VAR_GLOBAL
	DAU : ARRAY [1..100] OF DAU; //Instantiate 100 DAU's  This can be made higher if we think that 1 system will ever have more than 100 DAU's
END_VAR

(* stored: Version 1.1.0.1, ProductVersion 3.1.4022.12
   GVL GVL_DUA: Id {964d5aa3-6374-4cdb-97c1-b235e9795180} *)
